# EPICS substitutions: n1912a/Db/n1912a.substitutions
file "n1912a-gen.template" { pattern
{}
{}
}

#file "n1912a-chan.template" { pattern
#{CHAN}
#{01}
#{02}
#}
